Staubli VAL3: ack.pgx

public program ack(num x_nHeaderTime, num x_nElapsedTime)
begin

  // Do nothing
  // See start() program for more details

end
